(* Logix 5000 project; controller LeakTestAuto vendor 1 type 14 code 226 rev 37.11; software revision 37.01; part 6 of 13 *)
(* tags used below, declared in another part *)
   AOI_CTS1 : AOI_CTS_INSTRUMENT;
   AOI_OP220_HomingSeq : AOI_Sequencer_x64;
   AOI_OP220_Seq : AOI_Sequencer_x64;
   AOI_RobotPos : AOI_RobotPositions;
   AOI_SeqSteps : AOI_StandardSeqSteps;
   AOI_SRX100 : AOI_KeyenceBarcode;
   Barcode_ResultData : STR_Barcode;
   BarcodeBypass : BOOL;
   BarcodeInputs : udt_KeyenceScannerInputs;
   BarcodeScanner : udt_OutputStructure;
   Config_ConveyorHomeCounter : DINT;
   Config_ConveyorHomeCounterEnter : BOOL;
   Config_CylinderWaitTime : DINT;
   Config_CylinderWaitTimeEnter : BOOL;
   Config_MaxFailCount : DINT;
   Config_MaxFailCountEnter : BOOL;
   Conveyor : udt_OutputStructure;
   Conveyor_Seq : udt_SequenceStructure_X64;
   ConveyorHomeCounter : COUNTER;
   CTS1_BarcodeWrite : STRING80;
   CTS2_BarcodeWrite : STRING80;
   CurrentDUTData : udt_DUTHistory[2];
   DryCycle_N1Ready : BOOL;
   DryCycle_N2Ready : BOOL;
   FailCount : COUNTER;
   HomingClearNestsBypass : BOOL;
   InfeedCounter : COUNTER;
   LeakTester1 : udt_OutputStructure;
   LeakTester2 : udt_OutputStructure;
   Mode_CapCTS : BOOL;
   Nest1Bypass : BOOL;
   Nest1Cylinder : udt_OutputStructure;
   Nest1Empty : BOOL;
   Nest1Ready : BOOL;
   Nest2Bypass : BOOL;
   Nest2Cylinder : udt_OutputStructure;
   Nest2Empty : BOOL;
   Nest2Ready : BOOL;
   ONS_FailBinRemoved : BOOL;
   OP220 : udt_Mode;
   OP220_HomingSeq : udt_SequenceStructure_X64;
   OP220_Seq : udt_SequenceStructure_X64;
   OutfeedCounter : COUNTER;
   ResetFeedCounters : BOOL;
   RFID_CmdNest1 : BOOL;
   RFID_CmdNest2 : BOOL;
   RFID_Nest2Delay : TIMER;
   RFID_RWHAllPort : RWH_CMD;
   RFID_TagStatus : BOOL[32];
   RFIDBypass : BOOL;
   RFIDScanner : udt_OutputStructure;
   Robot : udt_OutputStructure;
   RobotGripper : udt_OutputStructure;
   RobotInputs : udt_EpsonInputs;
   RobotOutputs : udt_EpsonOutputs;
   TON_ConvUnloadDelay : TIMER;
   TON_FailChute : TIMER[10];
   TON_Nest1DryCycleDryTest : TIMER;
   TON_Nest2DryCycleDryTest : TIMER;
   I_OP220_N3_CONVEYOR_UNLOAD : ALIAS FOR Local:3:I.Pt14.Data;
   I_OP220_N3_DUT_PRE_NEST_0 : ALIAS FOR Local:3:I.Pt00.Data;
   I_OP220_N3_DUT_PRE_NEST_1 : ALIAS FOR Local:3:I.Pt01.Data;
   I_OP220_N3_DUT_PRE_NEST_2 : ALIAS FOR Local:3:I.Pt02.Data;
   I_OP220_N3_NEST1_EXTEND : ALIAS FOR Local:3:I.Pt04.Data;
   I_OP220_N3_NEST1_HOME : ALIAS FOR Local:3:I.Pt03.Data;
   I_OP220_N3_NEST2_EXTEND : ALIAS FOR Local:3:I.Pt06.Data;
   I_OP220_N3_NEST2_HOME : ALIAS FOR Local:3:I.Pt05.Data;
   I_OP220_N3_REJECT_BIN_OK : ALIAS FOR Local:3:I.Pt09.Data;
   I_OP220_N3_REJECT_CHUTE_PART : ALIAS FOR Local:3:I.Pt10.Data;
   James_Dint : DINT;   // James Test Word
   O_OP220_N5_CONV_REV : ALIAS FOR Local:5:O.Pt11.Data;
   O_OP220_N5_EN_MAIN_AIR : ALIAS FOR Local:5:O.Pt04.Data;
   O_OP220_N5_EN_ROBOT_LATCHOFF : ALIAS FOR Local:5:O.Pt09.Data;
   PLC : AOI_PLC;
   ST1_Ignition_SerialNum : STRING;
   ST2_Ignition_SerialNum : STRING;
(* MainProgram, continued *)

ROUTINE R06_IOControl   (* ladder *)
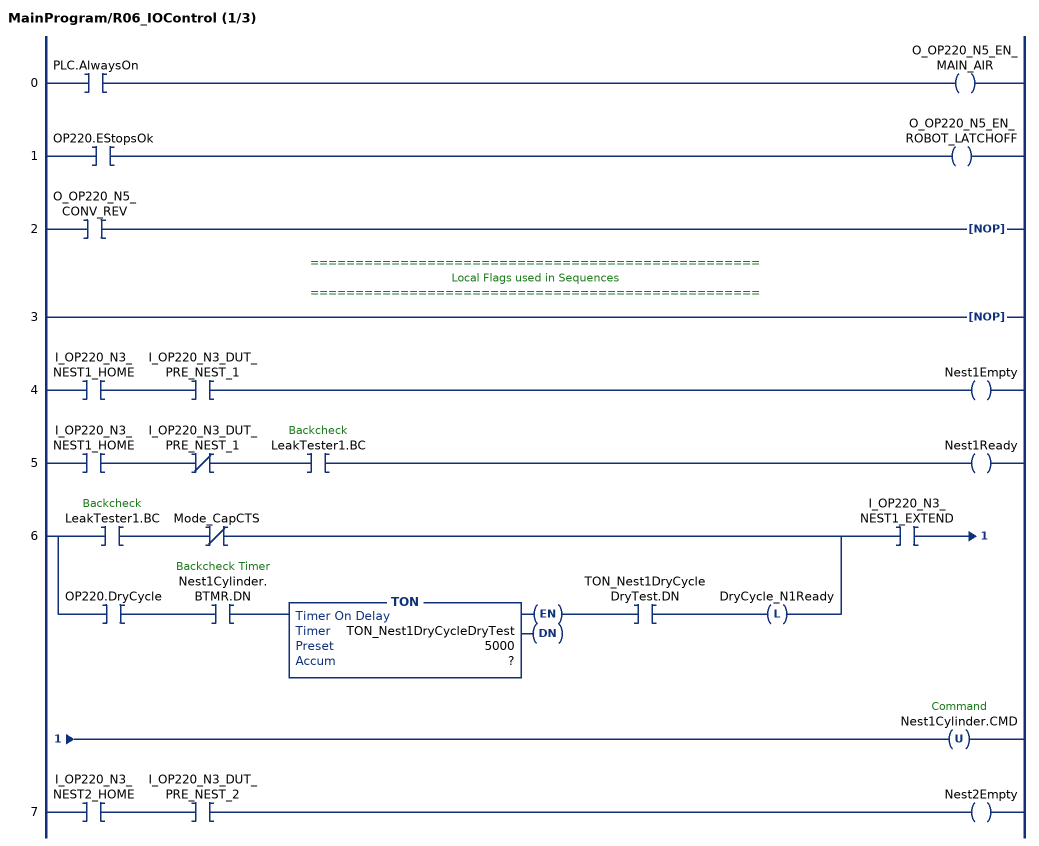
   0: XIC(PLC.AlwaysOn)OTE(O_OP220_N5_EN_MAIN_AIR);
   1: XIC(OP220.EStopsOk)OTE(O_OP220_N5_EN_ROBOT_LATCHOFF);
   2: XIC(O_OP220_N5_CONV_REV)NOP();
   // ==================================================
   // Local Flags used in Sequences
   // ==================================================
   3: NOP();
   4: XIC(I_OP220_N3_NEST1_HOME)XIC(I_OP220_N3_DUT_PRE_NEST_1)OTE(Nest1Empty);
   5: XIC(I_OP220_N3_NEST1_HOME)XIO(I_OP220_N3_DUT_PRE_NEST_1)XIC(LeakTester1.BC)OTE(Nest1Ready);
   6: [XIC(LeakTester1.BC) XIO(Mode_CapCTS) ,XIC(OP220.DryCycle) XIC(Nest1Cylinder.BTMR.DN) TON(TON_Nest1DryCycleDryTest,?,?) XIC(TON_Nest1DryCycleDryTest.DN) OTL(DryCycle_N1Ready) ]XIC(I_OP220_N3_NEST1_EXTEND)OTU(Nest1Cylinder.CMD);
   7: XIC(I_OP220_N3_NEST2_HOME)XIC(I_OP220_N3_DUT_PRE_NEST_2)OTE(Nest2Empty);
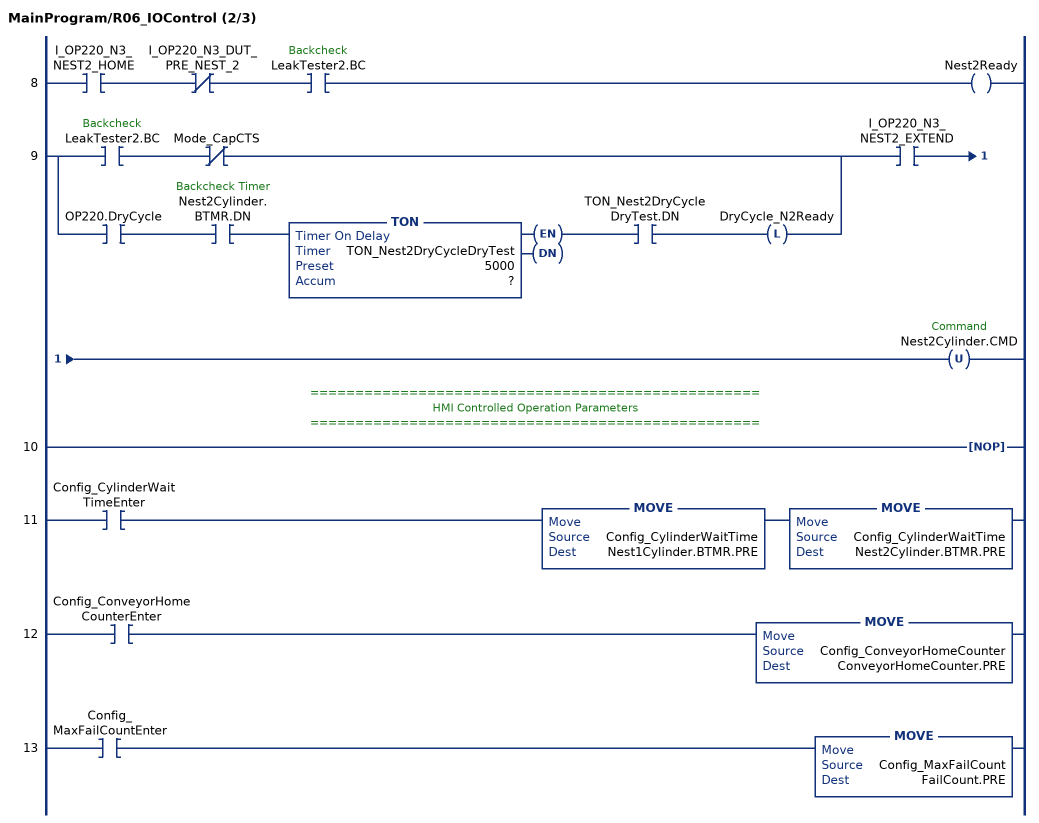
   8: XIC(I_OP220_N3_NEST2_HOME)XIO(I_OP220_N3_DUT_PRE_NEST_2)XIC(LeakTester2.BC)OTE(Nest2Ready);
   9: [XIC(LeakTester2.BC) XIO(Mode_CapCTS) ,XIC(OP220.DryCycle) XIC(Nest2Cylinder.BTMR.DN) TON(TON_Nest2DryCycleDryTest,?,?) XIC(TON_Nest2DryCycleDryTest.DN) OTL(DryCycle_N2Ready) ]XIC(I_OP220_N3_NEST2_EXTEND)OTU(Nest2Cylinder.CMD);
   // ==================================================
   // HMI Controlled Operation Parameters
   // ==================================================
   10: NOP();
   11: XIC(Config_CylinderWaitTimeEnter)MOVE(Config_CylinderWaitTime,Nest1Cylinder.BTMR.PRE)MOVE(Config_CylinderWaitTime,Nest2Cylinder.BTMR.PRE);
   12: XIC(Config_ConveyorHomeCounterEnter)MOVE(Config_ConveyorHomeCounter,ConveyorHomeCounter.PRE);
   13: XIC(Config_MaxFailCountEnter)MOVE(Config_MaxFailCount,FailCount.PRE);
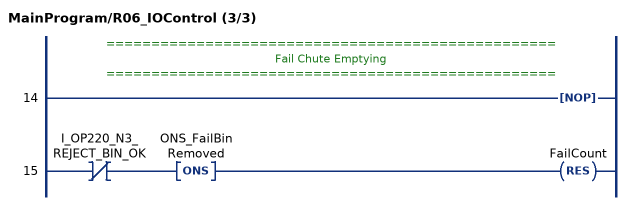
   // ==================================================
   // Fail Chute Emptying
   // ==================================================
   14: NOP();
   15: XIO(I_OP220_N3_REJECT_BIN_OK)ONS(ONS_FailBinRemoved)RES(FailCount);
END_ROUTINE

ROUTINE R09_Homing   (* ladder *)
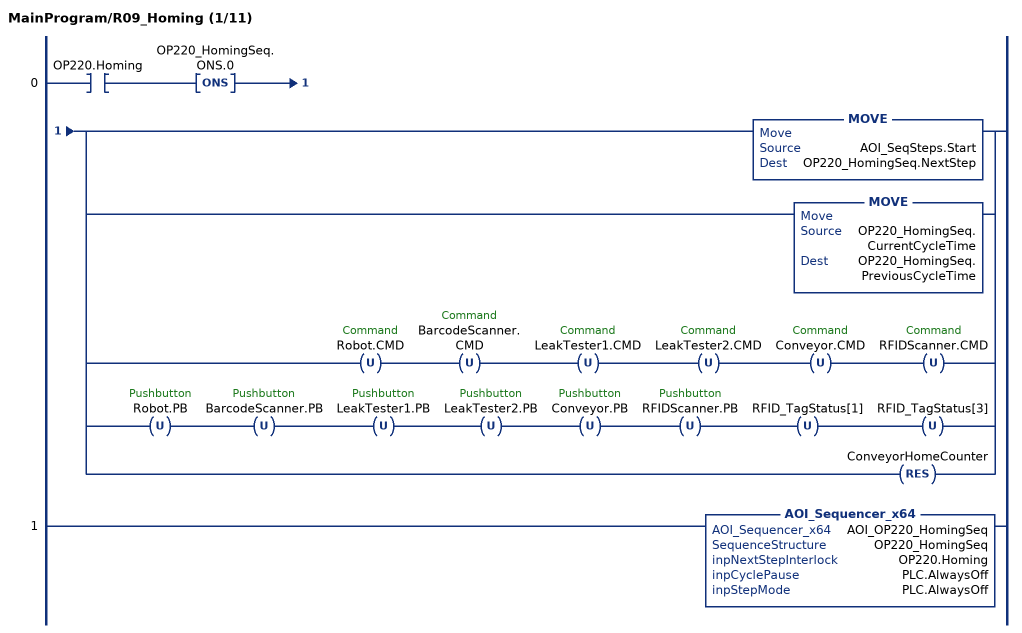
   0: XIC(OP220.Homing)ONS(OP220_HomingSeq.ONS.0)[MOVE(AOI_SeqSteps.Start,OP220_HomingSeq.NextStep) ,MOVE(OP220_HomingSeq.CurrentCycleTime,OP220_HomingSeq.PreviousCycleTime) ,OTU(Robot.CMD) OTU(BarcodeScanner.CMD) OTU(LeakTester1.CMD) OTU(LeakTester2.CMD) OTU(Conveyor.CMD) OTU(RFIDScanner.CMD) ,OTU(Robot.PB) OTU(BarcodeScanner.PB) OTU(LeakTester1.PB) OTU(LeakTester2.PB) OTU(Conveyor.PB) OTU(RFIDScanner.PB) OTU(RFID_TagStatus[1]) OTU(RFID_TagStatus[3]) ,RES(ConveyorHomeCounter) ];
   1: AOI_Sequencer_x64(AOI_OP220_HomingSeq,OP220_HomingSeq,OP220.Homing,PLC.AlwaysOff,PLC.AlwaysOff);
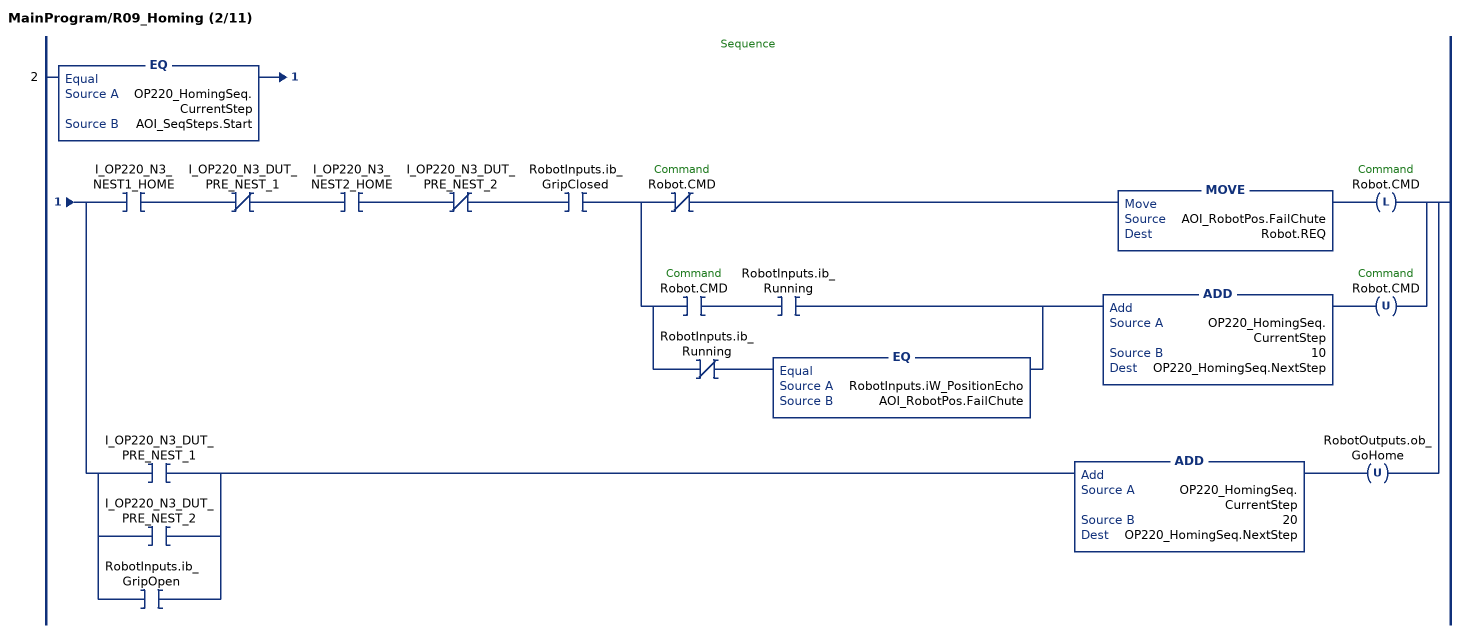
   // Sequence
   2: EQ(OP220_HomingSeq.CurrentStep,AOI_SeqSteps.Start)[XIC(I_OP220_N3_NEST1_HOME) XIO(I_OP220_N3_DUT_PRE_NEST_1) XIC(I_OP220_N3_NEST2_HOME) XIO(I_OP220_N3_DUT_PRE_NEST_2) XIC(RobotInputs.ib_GripClosed) [XIO(Robot.CMD) MOVE(AOI_RobotPos.FailChute,Robot.REQ) OTL(Robot.CMD) ,[XIC(Robot.CMD) XIC(RobotInputs.ib_Running) ,XIO(RobotInputs.ib_Running) EQ(RobotInputs.iW_PositionEcho,AOI_RobotPos.FailChute) ] ADD(OP220_HomingSeq.CurrentStep,10,OP220_HomingSeq.NextStep) OTU(Robot.CMD) ] ,[XIC(I_OP220_N3_DUT_PRE_NEST_1) ,XIC(I_OP220_N3_DUT_PRE_NEST_2) ,XIC(RobotInputs.ib_GripOpen) ] ADD(OP220_HomingSeq.CurrentStep,20,OP220_HomingSeq.NextStep) OTU(RobotOutputs.ob_GoHome) ];
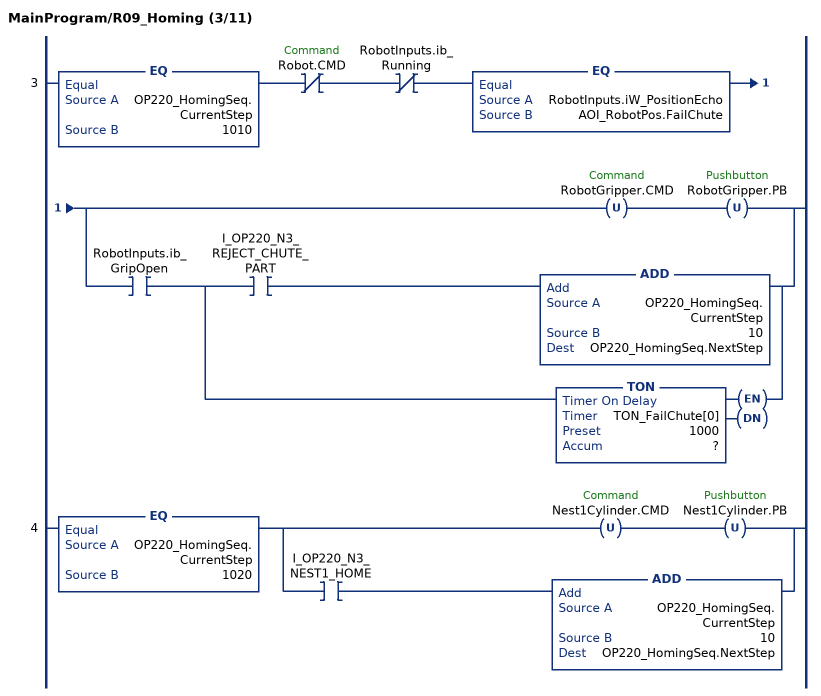
   3: EQ(OP220_HomingSeq.CurrentStep,1010)XIO(Robot.CMD)XIO(RobotInputs.ib_Running)EQ(RobotInputs.iW_PositionEcho,AOI_RobotPos.FailChute)[OTU(RobotGripper.CMD) OTU(RobotGripper.PB) ,XIC(RobotInputs.ib_GripOpen) [XIC(I_OP220_N3_REJECT_CHUTE_PART) ADD(OP220_HomingSeq.CurrentStep,10,OP220_HomingSeq.NextStep) ,TON(TON_FailChute[0],?,?) ] ];
   4: EQ(OP220_HomingSeq.CurrentStep,1020)[OTU(Nest1Cylinder.CMD) OTU(Nest1Cylinder.PB) ,XIC(I_OP220_N3_NEST1_HOME) ADD(OP220_HomingSeq.CurrentStep,10,OP220_HomingSeq.NextStep) ];
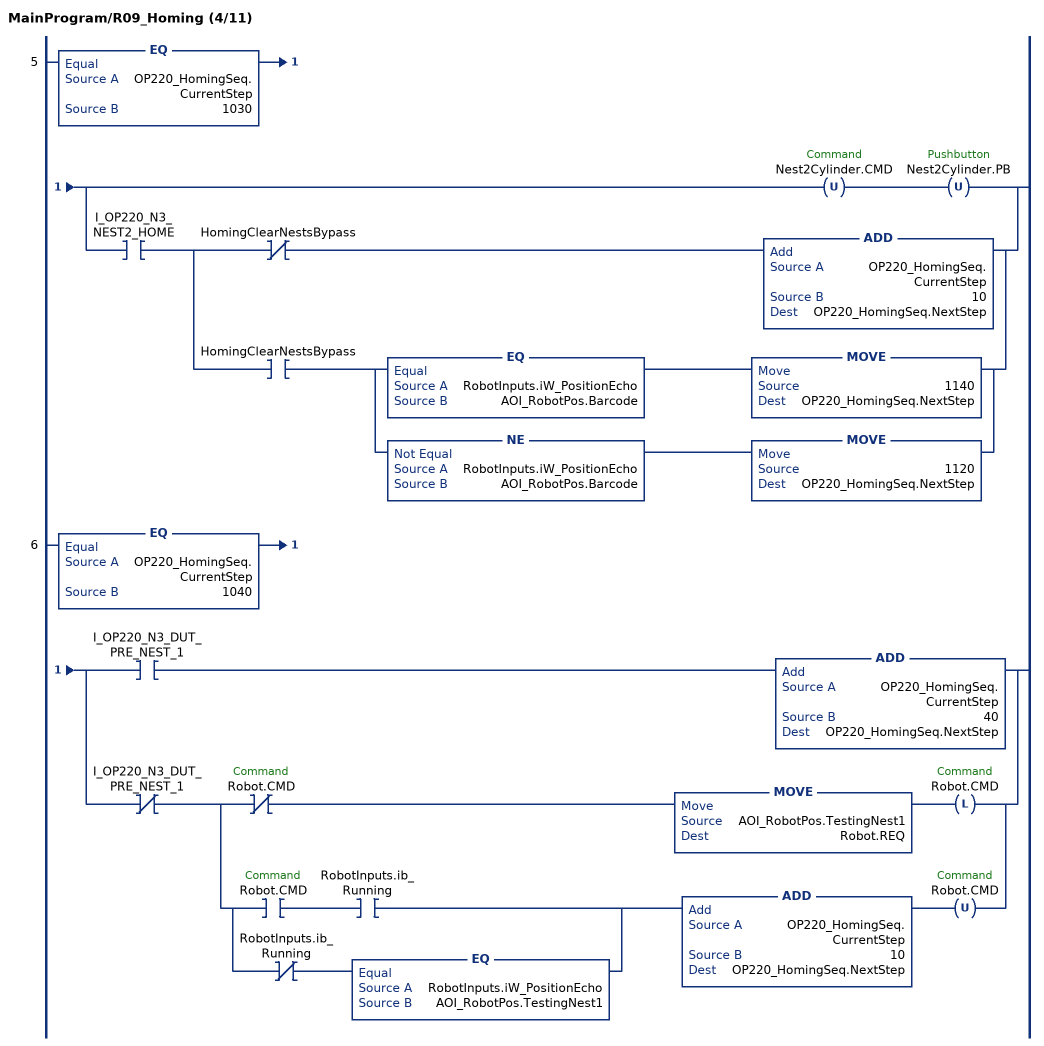
   5: EQ(OP220_HomingSeq.CurrentStep,1030)[OTU(Nest2Cylinder.CMD) OTU(Nest2Cylinder.PB) ,XIC(I_OP220_N3_NEST2_HOME) [XIO(HomingClearNestsBypass) ADD(OP220_HomingSeq.CurrentStep,10,OP220_HomingSeq.NextStep) ,XIC(HomingClearNestsBypass) [EQ(RobotInputs.iW_PositionEcho,AOI_RobotPos.Barcode) MOVE(1140,OP220_HomingSeq.NextStep) ,NE(RobotInputs.iW_PositionEcho,AOI_RobotPos.Barcode) MOVE(1120,OP220_HomingSeq.NextStep) ] ] ];
   6: EQ(OP220_HomingSeq.CurrentStep,1040)[XIC(I_OP220_N3_DUT_PRE_NEST_1) ADD(OP220_HomingSeq.CurrentStep,40,OP220_HomingSeq.NextStep) ,XIO(I_OP220_N3_DUT_PRE_NEST_1) [XIO(Robot.CMD) MOVE(AOI_RobotPos.TestingNest1,Robot.REQ) OTL(Robot.CMD) ,[XIC(Robot.CMD) XIC(RobotInputs.ib_Running) ,XIO(RobotInputs.ib_Running) EQ(RobotInputs.iW_PositionEcho,AOI_RobotPos.TestingNest1) ] ADD(OP220_HomingSeq.CurrentStep,10,OP220_HomingSeq.NextStep) OTU(Robot.CMD) ] ];
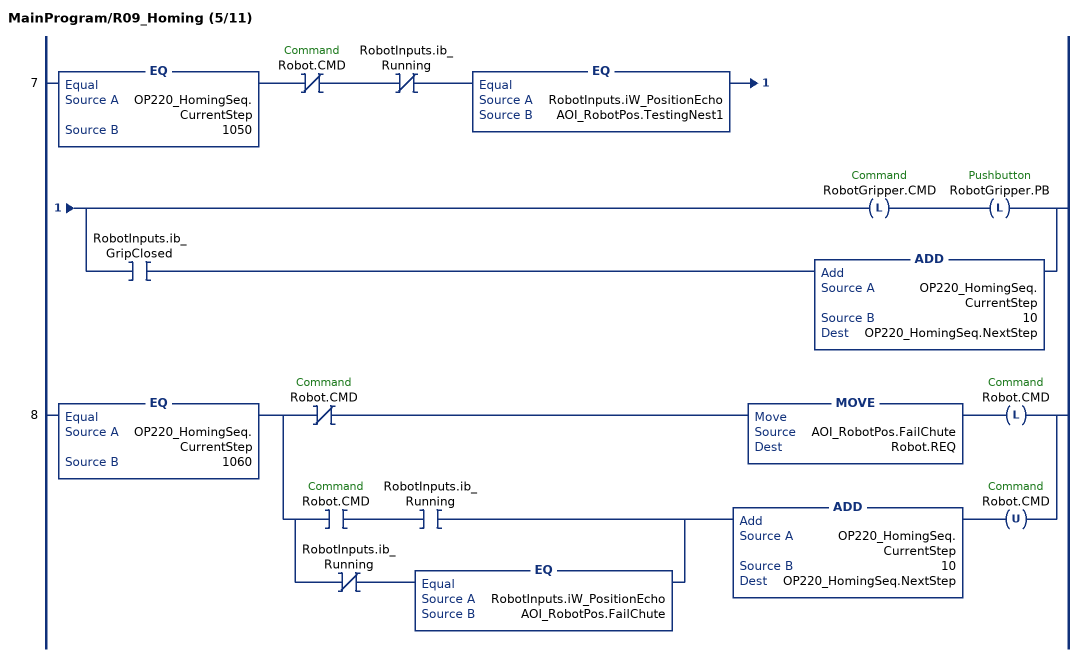
   7: EQ(OP220_HomingSeq.CurrentStep,1050)XIO(Robot.CMD)XIO(RobotInputs.ib_Running)EQ(RobotInputs.iW_PositionEcho,AOI_RobotPos.TestingNest1)[OTL(RobotGripper.CMD) OTL(RobotGripper.PB) ,XIC(RobotInputs.ib_GripClosed) ADD(OP220_HomingSeq.CurrentStep,10,OP220_HomingSeq.NextStep) ];
   8: EQ(OP220_HomingSeq.CurrentStep,1060)[XIO(Robot.CMD) MOVE(AOI_RobotPos.FailChute,Robot.REQ) OTL(Robot.CMD) ,[XIC(Robot.CMD) XIC(RobotInputs.ib_Running) ,XIO(RobotInputs.ib_Running) EQ(RobotInputs.iW_PositionEcho,AOI_RobotPos.FailChute) ] ADD(OP220_HomingSeq.CurrentStep,10,OP220_HomingSeq.NextStep) OTU(Robot.CMD) ];
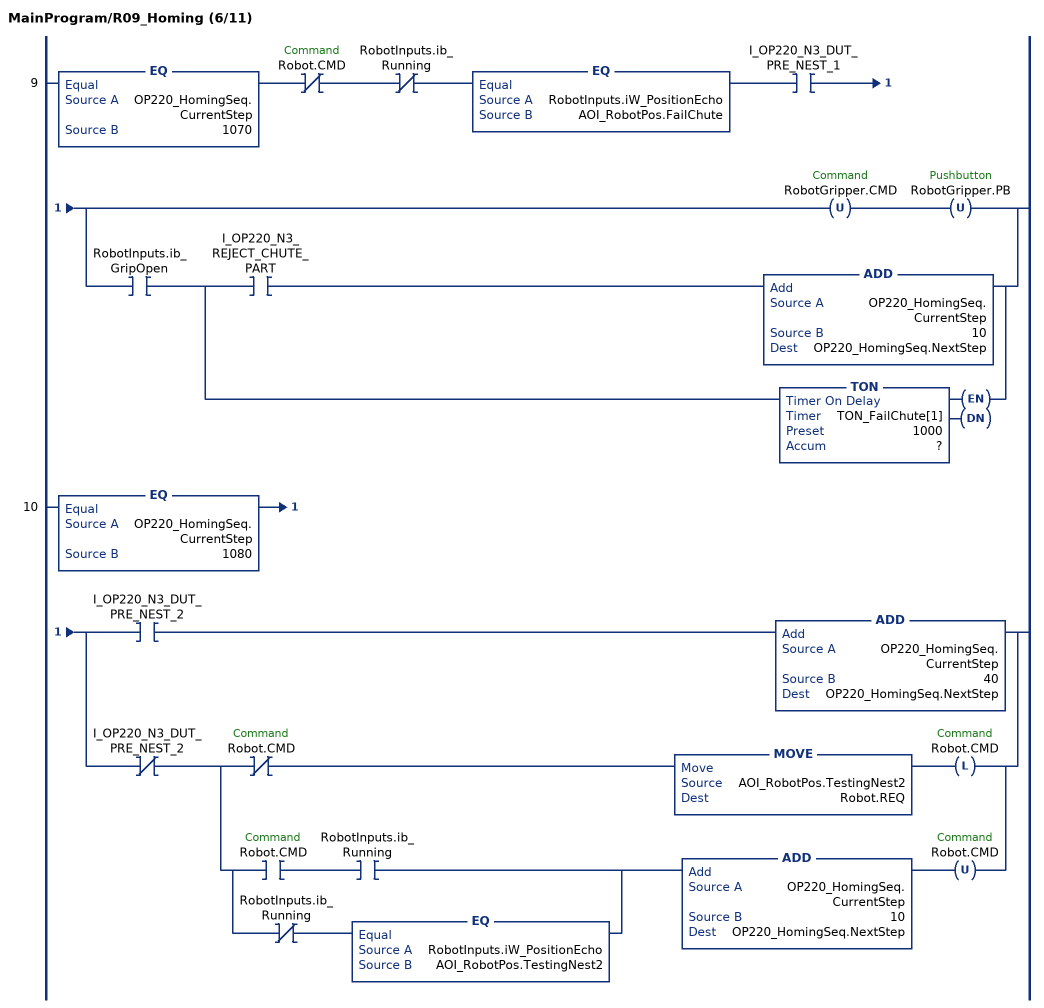
   9: EQ(OP220_HomingSeq.CurrentStep,1070)XIO(Robot.CMD)XIO(RobotInputs.ib_Running)EQ(RobotInputs.iW_PositionEcho,AOI_RobotPos.FailChute)XIC(I_OP220_N3_DUT_PRE_NEST_1)[OTU(RobotGripper.CMD) OTU(RobotGripper.PB) ,XIC(RobotInputs.ib_GripOpen) [XIC(I_OP220_N3_REJECT_CHUTE_PART) ADD(OP220_HomingSeq.CurrentStep,10,OP220_HomingSeq.NextStep) ,TON(TON_FailChute[1],?,?) ] ];
   10: EQ(OP220_HomingSeq.CurrentStep,1080)[XIC(I_OP220_N3_DUT_PRE_NEST_2) ADD(OP220_HomingSeq.CurrentStep,40,OP220_HomingSeq.NextStep) ,XIO(I_OP220_N3_DUT_PRE_NEST_2) [XIO(Robot.CMD) MOVE(AOI_RobotPos.TestingNest2,Robot.REQ) OTL(Robot.CMD) ,[XIC(Robot.CMD) XIC(RobotInputs.ib_Running) ,XIO(RobotInputs.ib_Running) EQ(RobotInputs.iW_PositionEcho,AOI_RobotPos.TestingNest2) ] ADD(OP220_HomingSeq.CurrentStep,10,OP220_HomingSeq.NextStep) OTU(Robot.CMD) ] ];
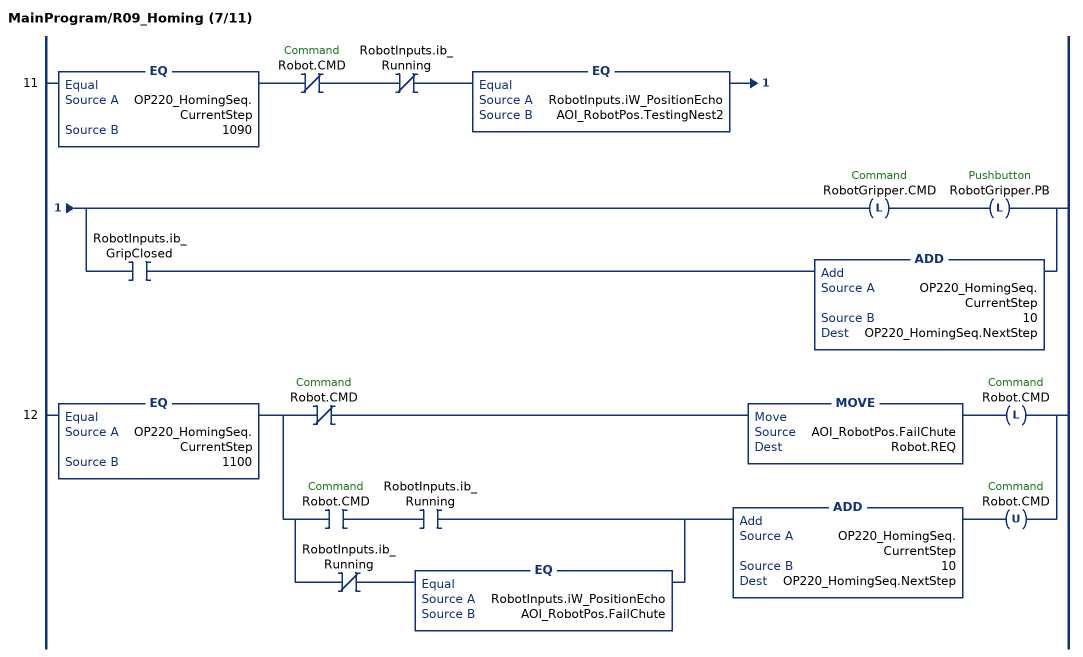
   11: EQ(OP220_HomingSeq.CurrentStep,1090)XIO(Robot.CMD)XIO(RobotInputs.ib_Running)EQ(RobotInputs.iW_PositionEcho,AOI_RobotPos.TestingNest2)[OTL(RobotGripper.CMD) OTL(RobotGripper.PB) ,XIC(RobotInputs.ib_GripClosed) ADD(OP220_HomingSeq.CurrentStep,10,OP220_HomingSeq.NextStep) ];
   12: EQ(OP220_HomingSeq.CurrentStep,1100)[XIO(Robot.CMD) MOVE(AOI_RobotPos.FailChute,Robot.REQ) OTL(Robot.CMD) ,[XIC(Robot.CMD) XIC(RobotInputs.ib_Running) ,XIO(RobotInputs.ib_Running) EQ(RobotInputs.iW_PositionEcho,AOI_RobotPos.FailChute) ] ADD(OP220_HomingSeq.CurrentStep,10,OP220_HomingSeq.NextStep) OTU(Robot.CMD) ];
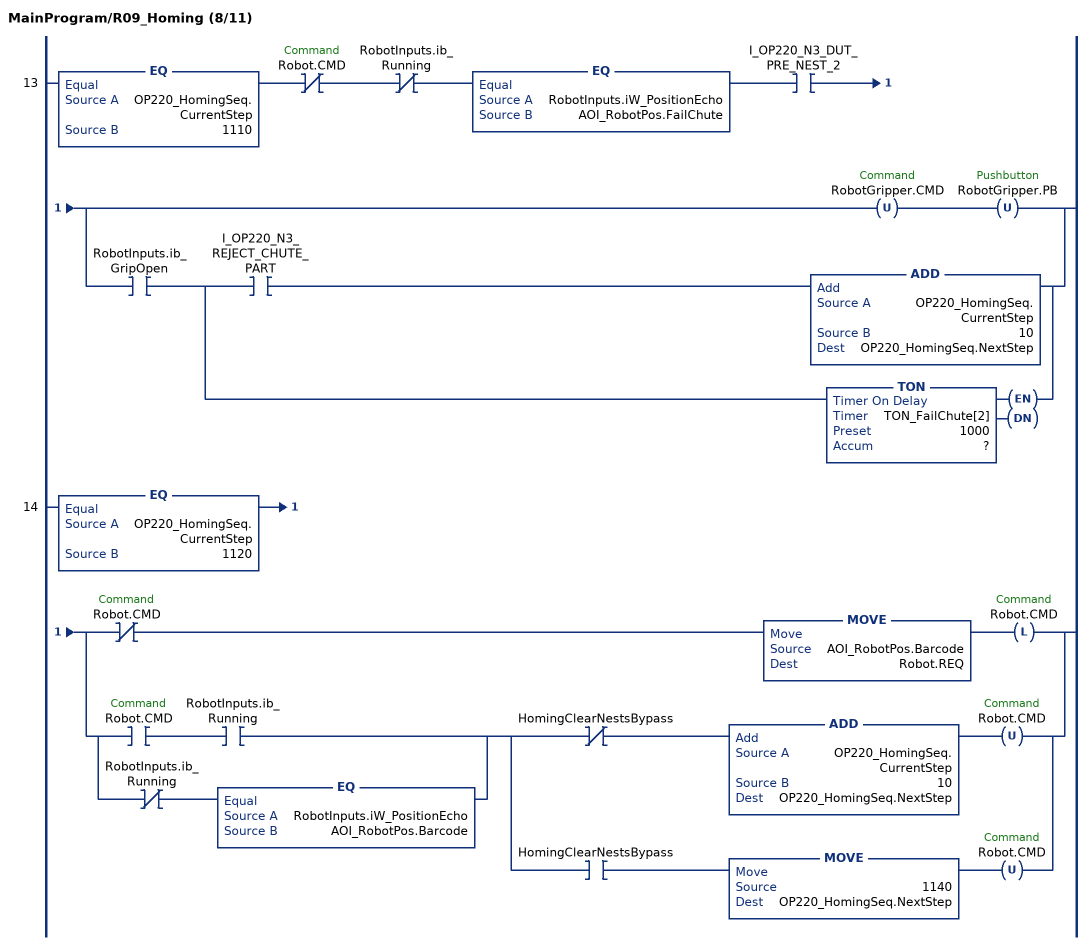
   13: EQ(OP220_HomingSeq.CurrentStep,1110)XIO(Robot.CMD)XIO(RobotInputs.ib_Running)EQ(RobotInputs.iW_PositionEcho,AOI_RobotPos.FailChute)XIC(I_OP220_N3_DUT_PRE_NEST_2)[OTU(RobotGripper.CMD) OTU(RobotGripper.PB) ,XIC(RobotInputs.ib_GripOpen) [XIC(I_OP220_N3_REJECT_CHUTE_PART) ADD(OP220_HomingSeq.CurrentStep,10,OP220_HomingSeq.NextStep) ,TON(TON_FailChute[2],?,?) ] ];
   14: EQ(OP220_HomingSeq.CurrentStep,1120)[XIO(Robot.CMD) MOVE(AOI_RobotPos.Barcode,Robot.REQ) OTL(Robot.CMD) ,[XIC(Robot.CMD) XIC(RobotInputs.ib_Running) ,XIO(RobotInputs.ib_Running) EQ(RobotInputs.iW_PositionEcho,AOI_RobotPos.Barcode) ] [XIO(HomingClearNestsBypass) ADD(OP220_HomingSeq.CurrentStep,10,OP220_HomingSeq.NextStep) OTU(Robot.CMD) ,XIC(HomingClearNestsBypass) MOVE(1140,OP220_HomingSeq.NextStep) OTU(Robot.CMD) ] ];
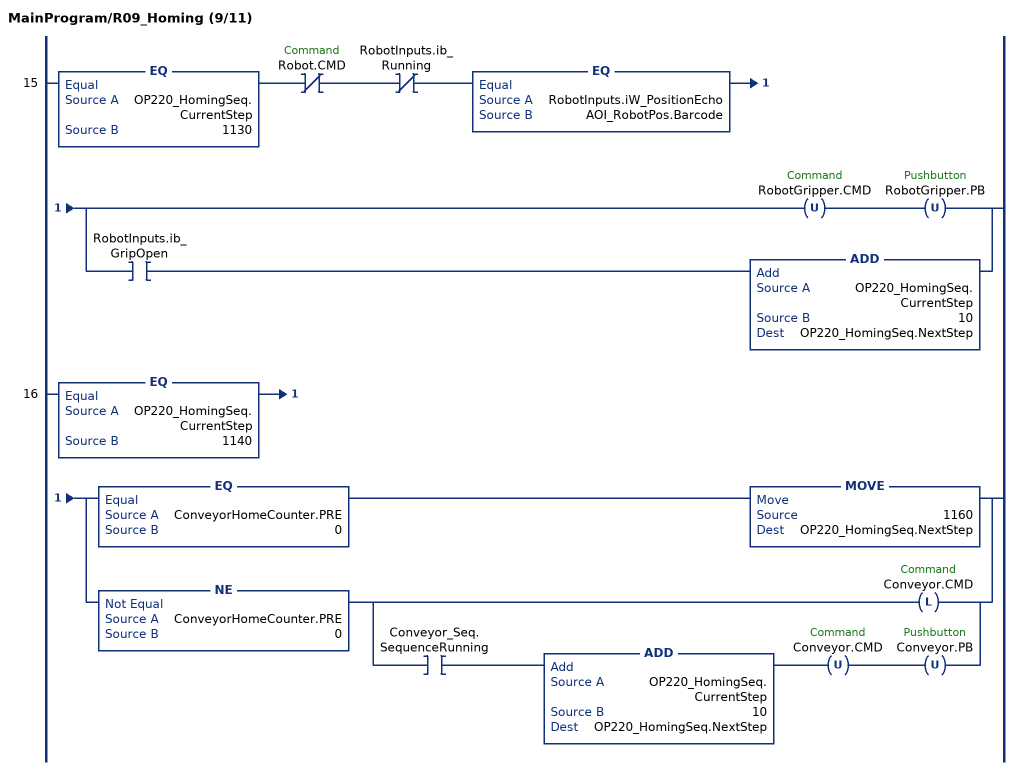
   15: EQ(OP220_HomingSeq.CurrentStep,1130)XIO(Robot.CMD)XIO(RobotInputs.ib_Running)EQ(RobotInputs.iW_PositionEcho,AOI_RobotPos.Barcode)[OTU(RobotGripper.CMD) OTU(RobotGripper.PB) ,XIC(RobotInputs.ib_GripOpen) ADD(OP220_HomingSeq.CurrentStep,10,OP220_HomingSeq.NextStep) ];
   16: EQ(OP220_HomingSeq.CurrentStep,1140)[EQ(ConveyorHomeCounter.PRE,0) MOVE(1160,OP220_HomingSeq.NextStep) ,NE(ConveyorHomeCounter.PRE,0) [OTL(Conveyor.CMD) ,XIC(Conveyor_Seq.SequenceRunning) ADD(OP220_HomingSeq.CurrentStep,10,OP220_HomingSeq.NextStep) OTU(Conveyor.CMD) OTU(Conveyor.PB) ] ];
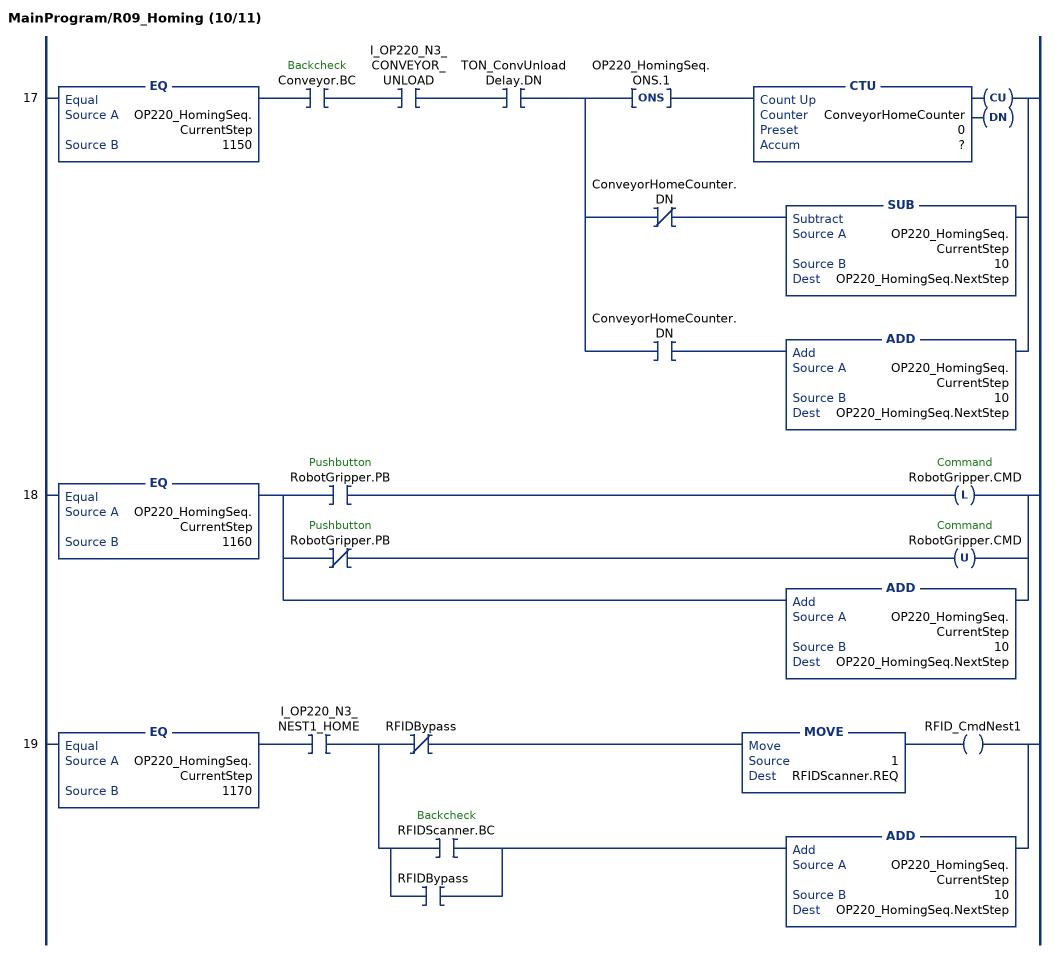
   17: EQ(OP220_HomingSeq.CurrentStep,1150)XIC(Conveyor.BC)XIC(I_OP220_N3_CONVEYOR_UNLOAD)XIC(TON_ConvUnloadDelay.DN)[ONS(OP220_HomingSeq.ONS.1) CTU(ConveyorHomeCounter,?,?) ,[XIO(ConveyorHomeCounter.DN) SUB(OP220_HomingSeq.CurrentStep,10,OP220_HomingSeq.NextStep) ,XIC(ConveyorHomeCounter.DN) ADD(OP220_HomingSeq.CurrentStep,10,OP220_HomingSeq.NextStep) ] ];
   18: EQ(OP220_HomingSeq.CurrentStep,1160)[XIC(RobotGripper.PB) OTL(RobotGripper.CMD) ,XIO(RobotGripper.PB) OTU(RobotGripper.CMD) ,ADD(OP220_HomingSeq.CurrentStep,10,OP220_HomingSeq.NextStep) ];
   19: EQ(OP220_HomingSeq.CurrentStep,1170)XIC(I_OP220_N3_NEST1_HOME)[XIO(RFIDBypass) MOVE(1,RFIDScanner.REQ) OTE(RFID_CmdNest1) ,[XIC(RFIDScanner.BC) ,XIC(RFIDBypass) ] ADD(OP220_HomingSeq.CurrentStep,10,OP220_HomingSeq.NextStep) ];
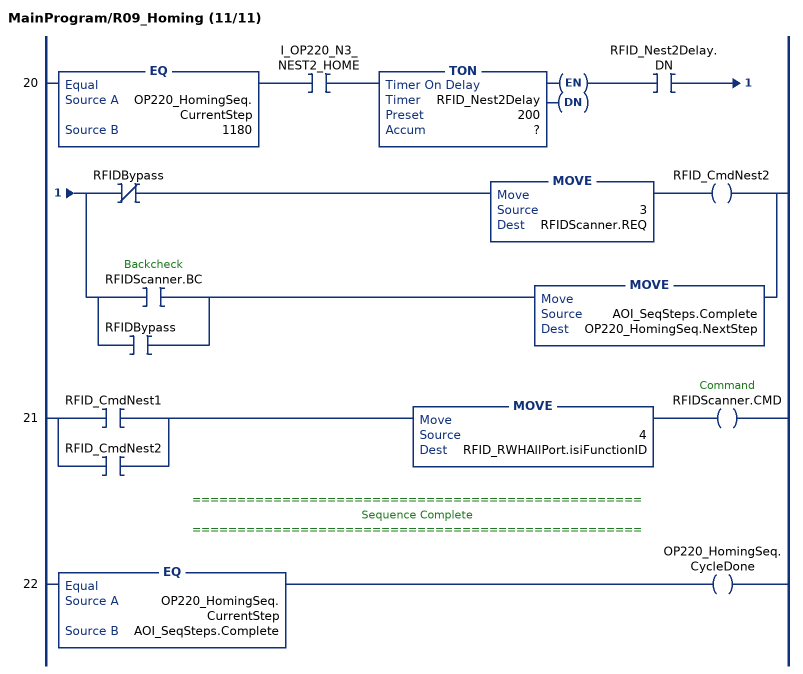
   20: EQ(OP220_HomingSeq.CurrentStep,1180)XIC(I_OP220_N3_NEST2_HOME)TON(RFID_Nest2Delay,?,?)XIC(RFID_Nest2Delay.DN)[XIO(RFIDBypass) MOVE(3,RFIDScanner.REQ) OTE(RFID_CmdNest2) ,[XIC(RFIDScanner.BC) ,XIC(RFIDBypass) ] MOVE(AOI_SeqSteps.Complete,OP220_HomingSeq.NextStep) ];
   21: [XIC(RFID_CmdNest1) ,XIC(RFID_CmdNest2) ]MOVE(4,RFID_RWHAllPort.isiFunctionID)OTE(RFIDScanner.CMD);
   // ==================================================
   // Sequence Complete
   // ==================================================
   22: EQ(OP220_HomingSeq.CurrentStep,AOI_SeqSteps.Complete)OTE(OP220_HomingSeq.CycleDone);
END_ROUTINE

ROUTINE R10_Sequence   (* ladder *)
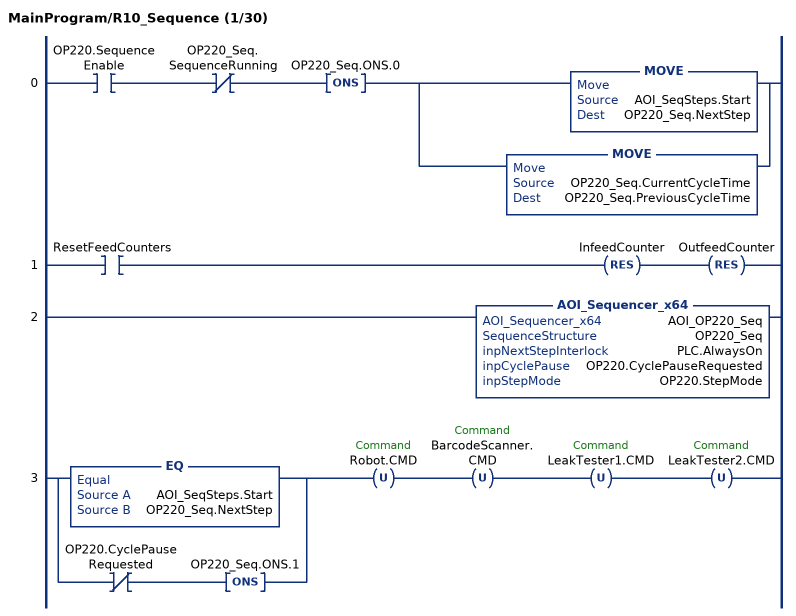
   0: XIC(OP220.SequenceEnable)XIO(OP220_Seq.SequenceRunning)ONS(OP220_Seq.ONS.0)[MOVE(AOI_SeqSteps.Start,OP220_Seq.NextStep) ,MOVE(OP220_Seq.CurrentCycleTime,OP220_Seq.PreviousCycleTime) ];
   1: XIC(ResetFeedCounters)RES(InfeedCounter)RES(OutfeedCounter);
   2: AOI_Sequencer_x64(AOI_OP220_Seq,OP220_Seq,PLC.AlwaysOn,OP220.CyclePauseRequested,OP220.StepMode);
   3: [EQ(AOI_SeqSteps.Start,OP220_Seq.NextStep) ,XIO(OP220.CyclePauseRequested) ONS(OP220_Seq.ONS.1) ]OTU(Robot.CMD)OTU(BarcodeScanner.CMD)OTU(LeakTester1.CMD)OTU(LeakTester2.CMD);
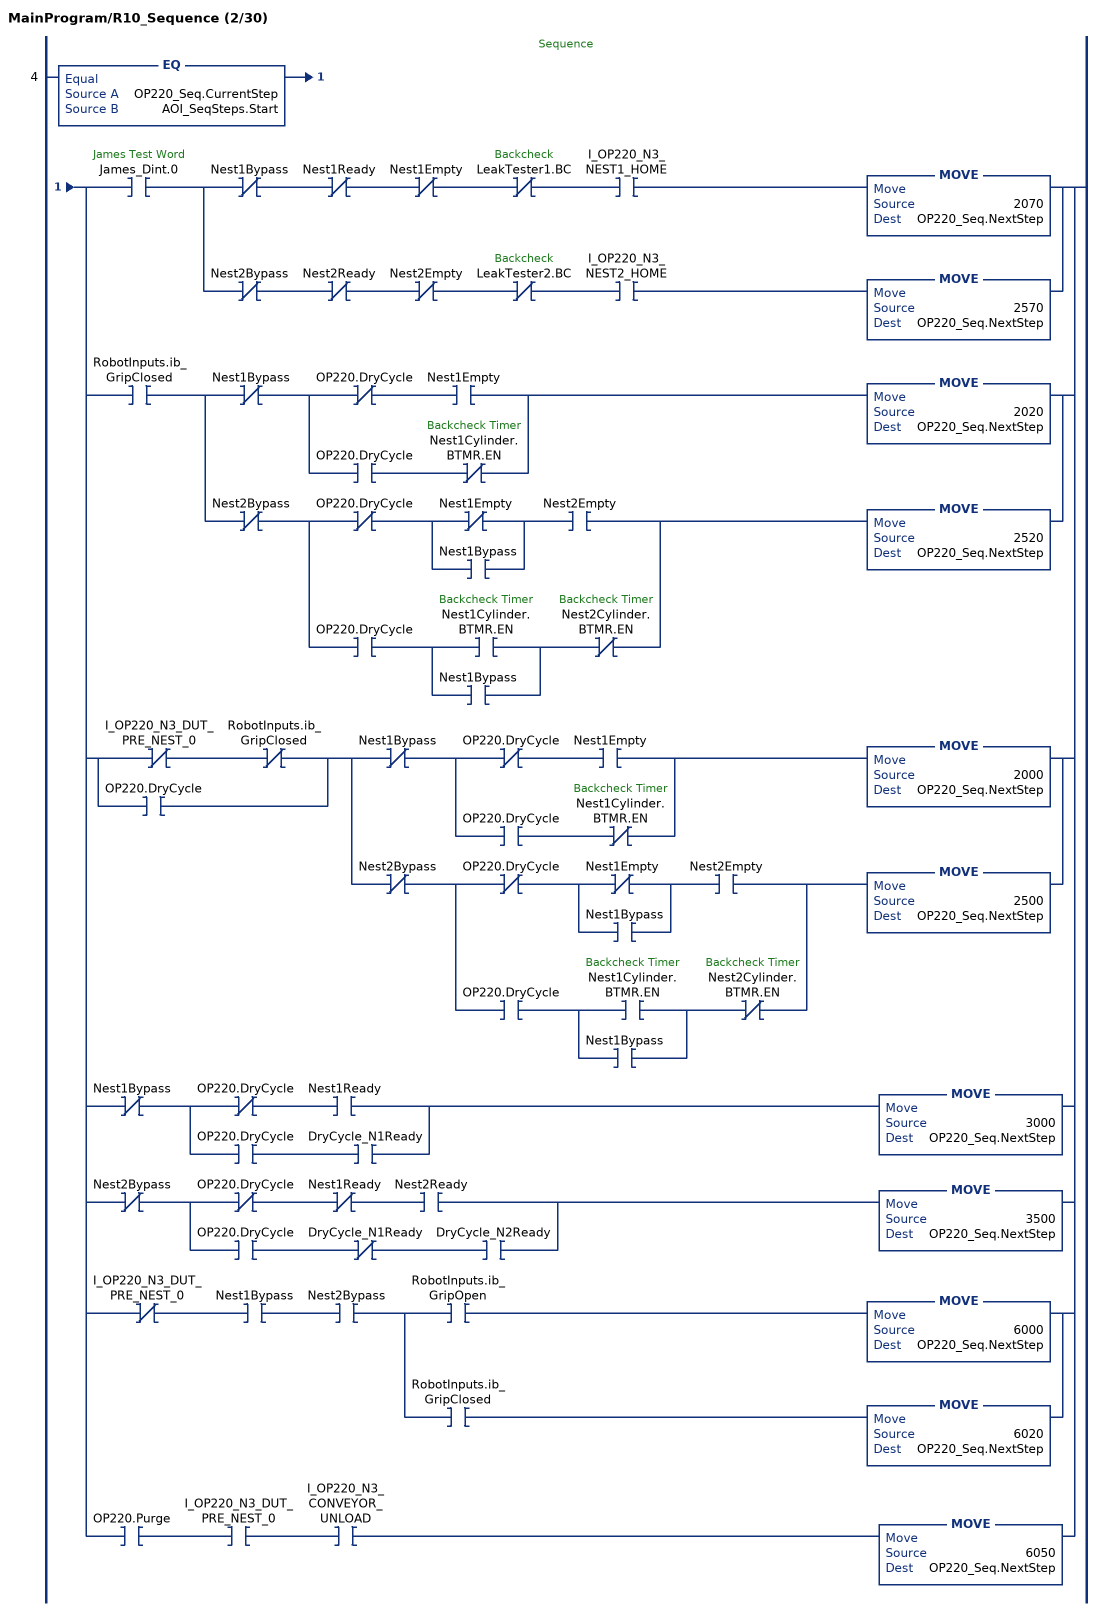
   // Sequence
   4: EQ(OP220_Seq.CurrentStep,AOI_SeqSteps.Start)[XIC(James_Dint.0) [XIO(Nest1Bypass) XIO(Nest1Ready) XIO(Nest1Empty) XIO(LeakTester1.BC) XIC(I_OP220_N3_NEST1_HOME) MOVE(2070,OP220_Seq.NextStep) ,XIO(Nest2Bypass) XIO(Nest2Ready) XIO(Nest2Empty) XIO(LeakTester2.BC) XIC(I_OP220_N3_NEST2_HOME) MOVE(2570,OP220_Seq.NextStep) ] ,XIC(RobotInputs.ib_GripClosed) [XIO(Nest1Bypass) [XIO(OP220.DryCycle) XIC(Nest1Empty) ,XIC(OP220.DryCycle) XIO(Nest1Cylinder.BTMR.EN) ] MOVE(2020,OP220_Seq.NextStep) ,XIO(Nest2Bypass) [XIO(OP220.DryCycle) [XIO(Nest1Empty) ,XIC(Nest1Bypass) ] XIC(Nest2Empty) ,XIC(OP220.DryCycle) [XIC(Nest1Cylinder.BTMR.EN) ,XIC(Nest1Bypass) ] XIO(Nest2Cylinder.BTMR.EN) ] MOVE(2520,OP220_Seq.NextStep) ] ,[XIO(I_OP220_N3_DUT_PRE_NEST_0) XIO(RobotInputs.ib_GripClosed) ,XIC(OP220.DryCycle) ] [XIO(Nest1Bypass) [XIO(OP220.DryCycle) XIC(Nest1Empty) ,XIC(OP220.DryCycle) XIO(Nest1Cylinder.BTMR.EN) ] MOVE(2000,OP220_Seq.NextStep) ,XIO(Nest2Bypass) [XIO(OP220.DryCycle) [XIO(Nest1Empty) ,XIC(Nest1Bypass) ] XIC(Nest2Empty) ,XIC(OP220.DryCycle) [XIC(Nest1Cylinder.BTMR.EN) ,XIC(Nest1Bypass) ] XIO(Nest2Cylinder.BTMR.EN) ] MOVE(2500,OP220_Seq.NextStep) ] ,[XIO(Nest1Bypass) [XIO(OP220.DryCycle) XIC(Nest1Ready) ,XIC(OP220.DryCycle) XIC(DryCycle_N1Ready) ] MOVE(3000,OP220_Seq.NextStep) ,XIO(Nest2Bypass) [XIO(OP220.DryCycle) XIO(Nest1Ready) XIC(Nest2Ready) ,XIC(OP220.DryCycle) XIO(DryCycle_N1Ready) XIC(DryCycle_N2Ready) ] MOVE(3500,OP220_Seq.NextStep) ] ,XIO(I_OP220_N3_DUT_PRE_NEST_0) XIC(Nest1Bypass) XIC(Nest2Bypass) [XIC(RobotInputs.ib_GripOpen) MOVE(6000,OP220_Seq.NextStep) ,XIC(RobotInputs.ib_GripClosed) MOVE(6020,OP220_Seq.NextStep) ] ,XIC(OP220.Purge) XIC(I_OP220_N3_DUT_PRE_NEST_0) XIC(I_OP220_N3_CONVEYOR_UNLOAD) MOVE(6050,OP220_Seq.NextStep) ];
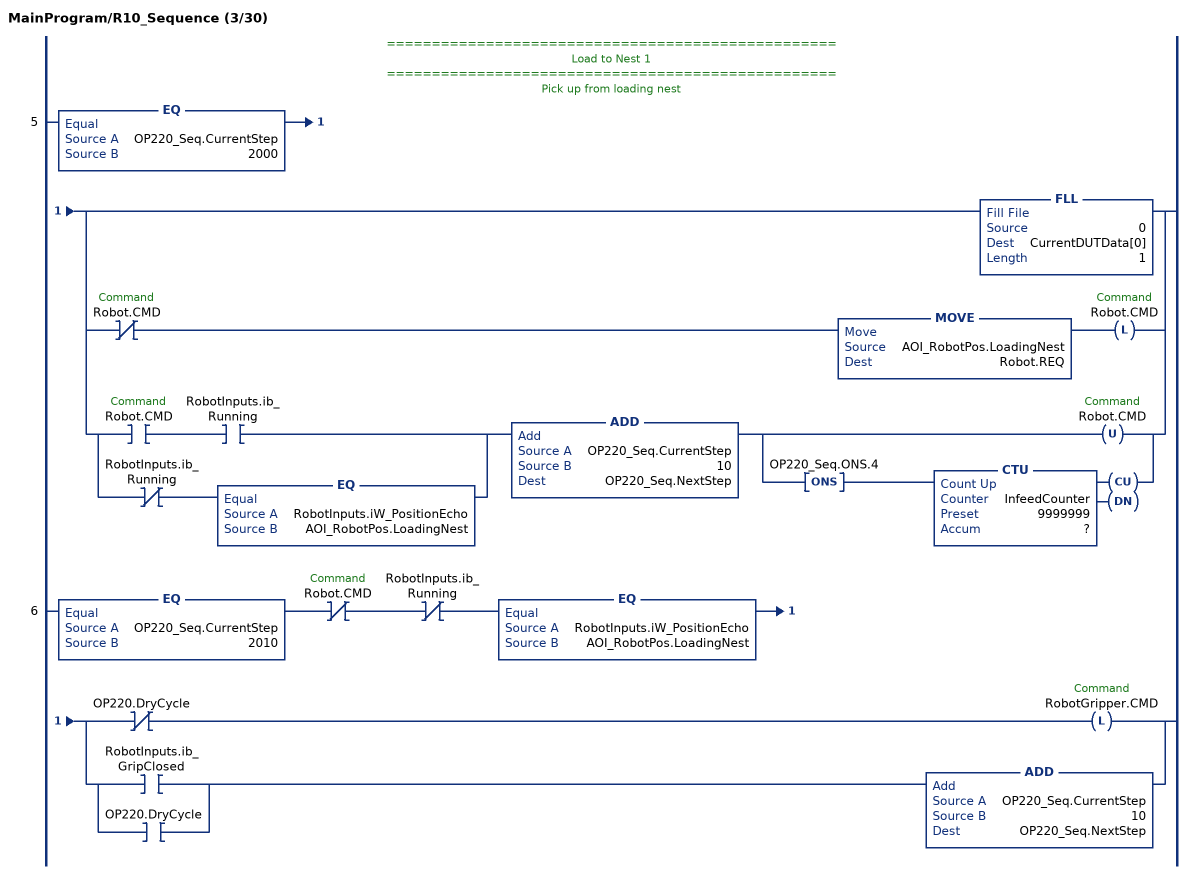
   // ==================================================
   // Load to Nest 1
   // ==================================================
   // Pick up from loading nest
   5: EQ(OP220_Seq.CurrentStep,2000)[FLL(0,CurrentDUTData[0],1) ,XIO(Robot.CMD) MOVE(AOI_RobotPos.LoadingNest,Robot.REQ) OTL(Robot.CMD) ,[XIC(Robot.CMD) XIC(RobotInputs.ib_Running) ,XIO(RobotInputs.ib_Running) EQ(RobotInputs.iW_PositionEcho,AOI_RobotPos.LoadingNest) ] ADD(OP220_Seq.CurrentStep,10,OP220_Seq.NextStep) [OTU(Robot.CMD) ,ONS(OP220_Seq.ONS.4) CTU(InfeedCounter,?,?) ] ];
   6: EQ(OP220_Seq.CurrentStep,2010)XIO(Robot.CMD)XIO(RobotInputs.ib_Running)EQ(RobotInputs.iW_PositionEcho,AOI_RobotPos.LoadingNest)[XIO(OP220.DryCycle) OTL(RobotGripper.CMD) ,[XIC(RobotInputs.ib_GripClosed) ,XIC(OP220.DryCycle) ] ADD(OP220_Seq.CurrentStep,10,OP220_Seq.NextStep) ];
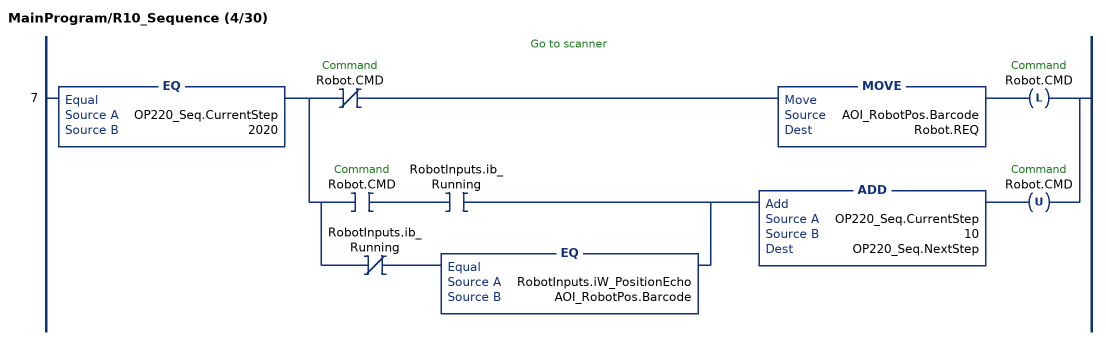
   // Go to scanner
   7: EQ(OP220_Seq.CurrentStep,2020)[XIO(Robot.CMD) MOVE(AOI_RobotPos.Barcode,Robot.REQ) OTL(Robot.CMD) ,[XIC(Robot.CMD) XIC(RobotInputs.ib_Running) ,XIO(RobotInputs.ib_Running) EQ(RobotInputs.iW_PositionEcho,AOI_RobotPos.Barcode) ] ADD(OP220_Seq.CurrentStep,10,OP220_Seq.NextStep) OTU(Robot.CMD) ];
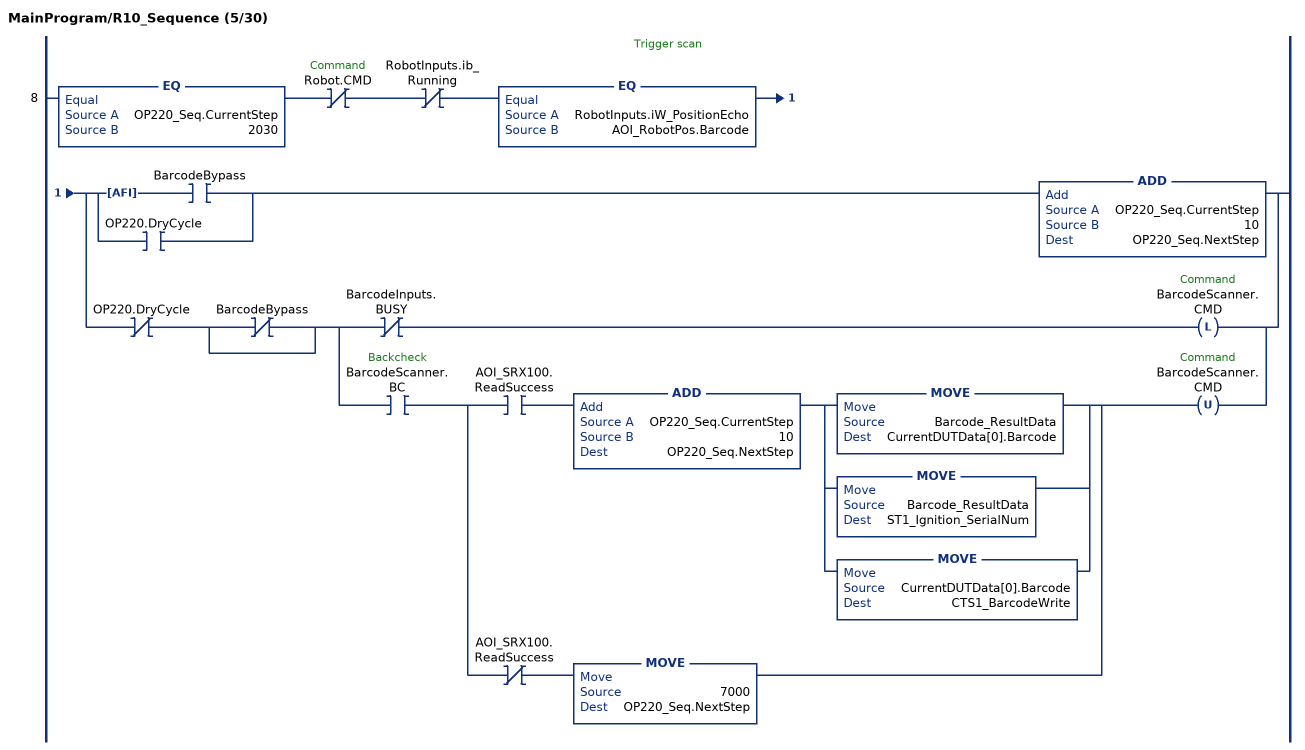
   // Trigger scan
   8: EQ(OP220_Seq.CurrentStep,2030)XIO(Robot.CMD)XIO(RobotInputs.ib_Running)EQ(RobotInputs.iW_PositionEcho,AOI_RobotPos.Barcode)[[AFI() XIC(BarcodeBypass) ,XIC(OP220.DryCycle) ] ADD(OP220_Seq.CurrentStep,10,OP220_Seq.NextStep) ,XIO(OP220.DryCycle) [XIO(BarcodeBypass) ,] [XIO(BarcodeInputs.BUSY) OTL(BarcodeScanner.CMD) ,XIC(BarcodeScanner.BC) [XIC(AOI_SRX100.ReadSuccess) ADD(OP220_Seq.CurrentStep,10,OP220_Seq.NextStep) [MOVE(Barcode_ResultData,CurrentDUTData[0].Barcode) ,[MOVE(Barcode_ResultData,ST1_Ignition_SerialNum) ,MOVE(CurrentDUTData[0].Barcode,CTS1_BarcodeWrite) ] ] ,XIO(AOI_SRX100.ReadSuccess) MOVE(7000,OP220_Seq.NextStep) ] OTU(BarcodeScanner.CMD) ] ];
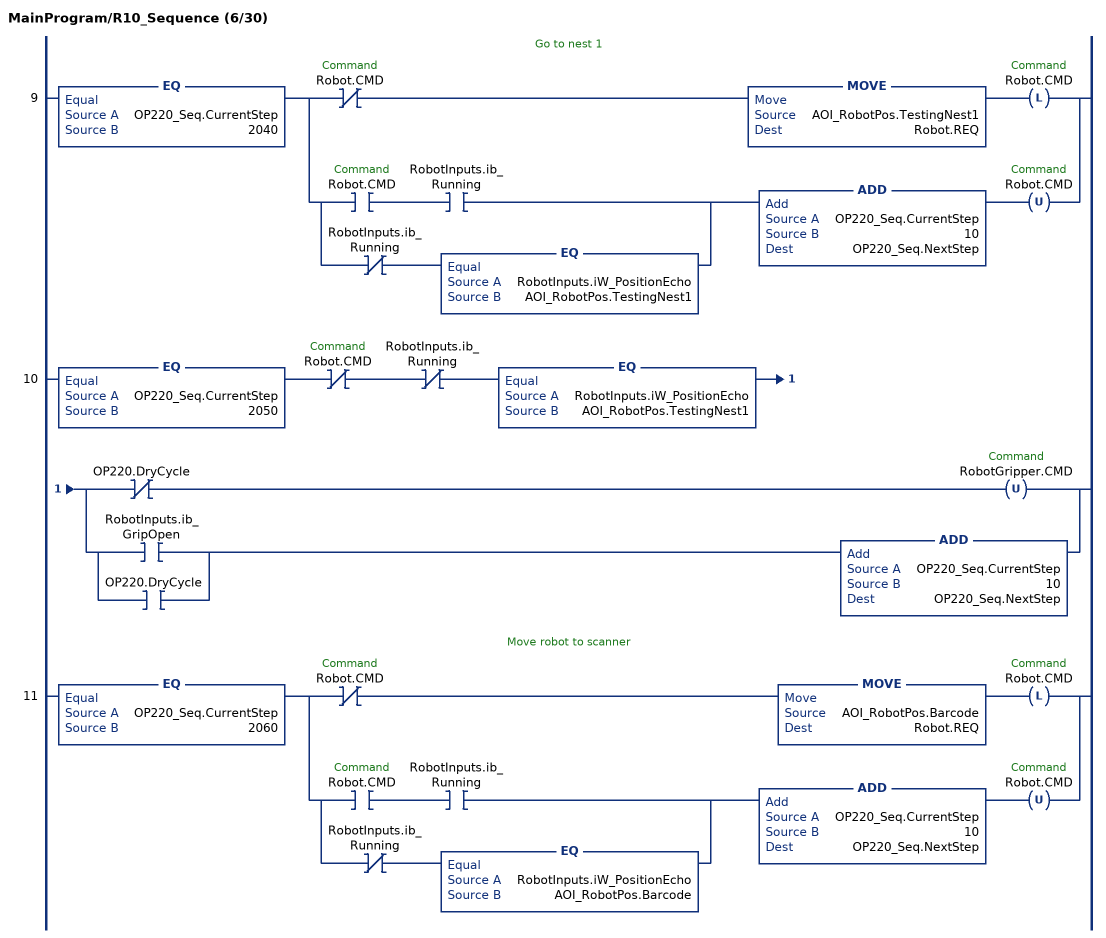
   // Go to nest 1
   9: EQ(OP220_Seq.CurrentStep,2040)[XIO(Robot.CMD) MOVE(AOI_RobotPos.TestingNest1,Robot.REQ) OTL(Robot.CMD) ,[XIC(Robot.CMD) XIC(RobotInputs.ib_Running) ,XIO(RobotInputs.ib_Running) EQ(RobotInputs.iW_PositionEcho,AOI_RobotPos.TestingNest1) ] ADD(OP220_Seq.CurrentStep,10,OP220_Seq.NextStep) OTU(Robot.CMD) ];
   10: EQ(OP220_Seq.CurrentStep,2050)XIO(Robot.CMD)XIO(RobotInputs.ib_Running)EQ(RobotInputs.iW_PositionEcho,AOI_RobotPos.TestingNest1)[XIO(OP220.DryCycle) OTU(RobotGripper.CMD) ,[XIC(RobotInputs.ib_GripOpen) ,XIC(OP220.DryCycle) ] ADD(OP220_Seq.CurrentStep,10,OP220_Seq.NextStep) ];
   // Move robot to scanner
   11: EQ(OP220_Seq.CurrentStep,2060)[XIO(Robot.CMD) MOVE(AOI_RobotPos.Barcode,Robot.REQ) OTL(Robot.CMD) ,[XIC(Robot.CMD) XIC(RobotInputs.ib_Running) ,XIO(RobotInputs.ib_Running) EQ(RobotInputs.iW_PositionEcho,AOI_RobotPos.Barcode) ] ADD(OP220_Seq.CurrentStep,10,OP220_Seq.NextStep) OTU(Robot.CMD) ];
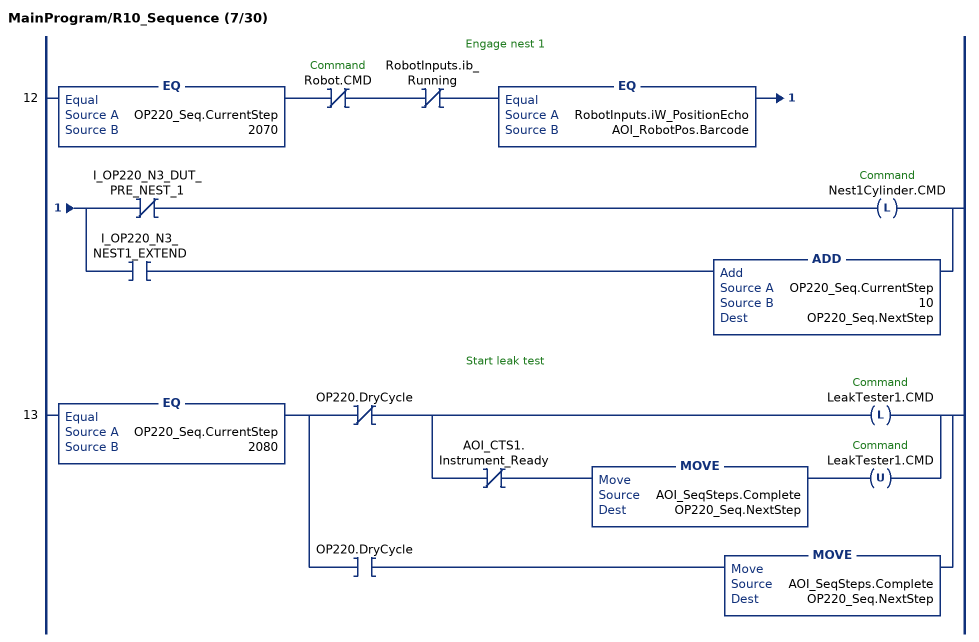
   // Engage nest 1
   12: EQ(OP220_Seq.CurrentStep,2070)XIO(Robot.CMD)XIO(RobotInputs.ib_Running)EQ(RobotInputs.iW_PositionEcho,AOI_RobotPos.Barcode)[XIO(I_OP220_N3_DUT_PRE_NEST_1) OTL(Nest1Cylinder.CMD) ,XIC(I_OP220_N3_NEST1_EXTEND) ADD(OP220_Seq.CurrentStep,10,OP220_Seq.NextStep) ];
   // Start leak test
   13: EQ(OP220_Seq.CurrentStep,2080)[XIO(OP220.DryCycle) [OTL(LeakTester1.CMD) ,XIO(AOI_CTS1.Instrument_Ready) MOVE(AOI_SeqSteps.Complete,OP220_Seq.NextStep) OTU(LeakTester1.CMD) ] ,XIC(OP220.DryCycle) MOVE(AOI_SeqSteps.Complete,OP220_Seq.NextStep) ];
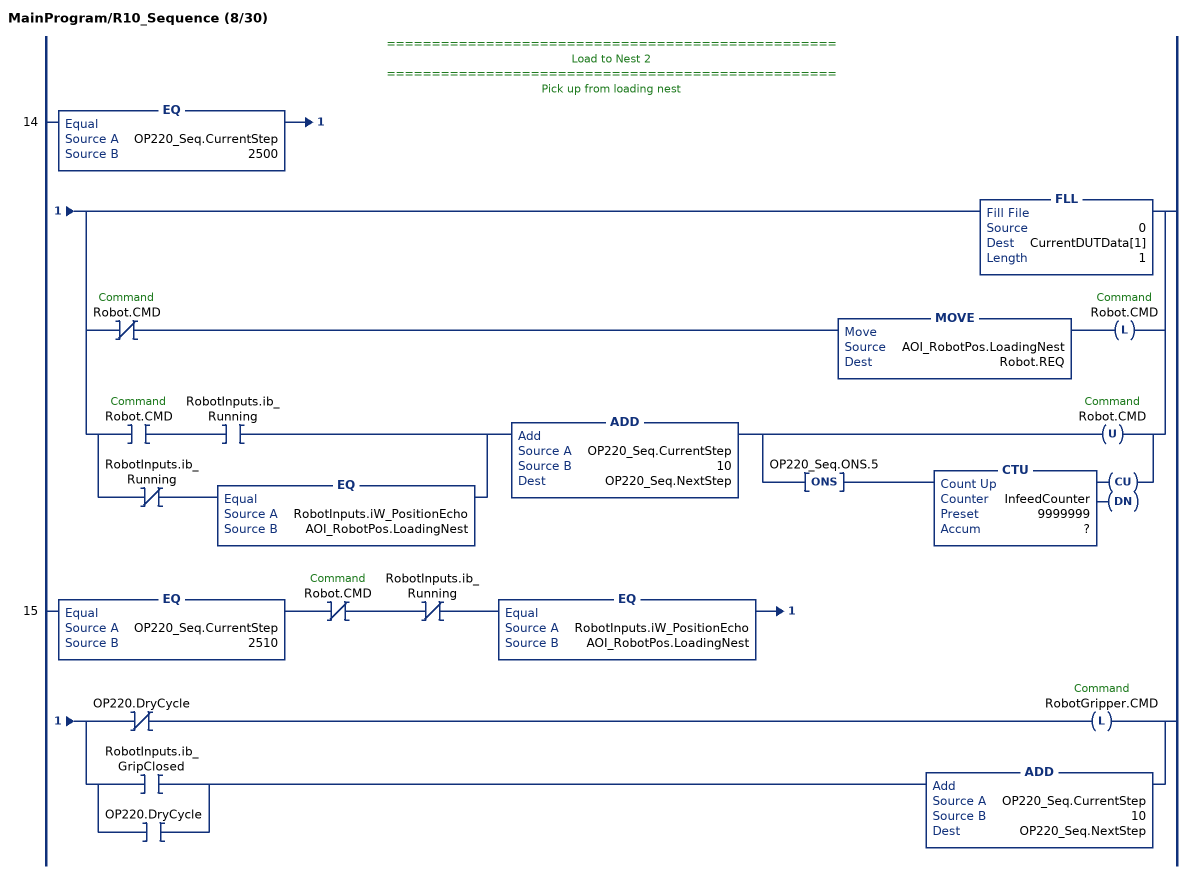
   // ==================================================
   // Load to Nest 2
   // ==================================================
   // Pick up from loading nest
   14: EQ(OP220_Seq.CurrentStep,2500)[FLL(0,CurrentDUTData[1],1) ,XIO(Robot.CMD) MOVE(AOI_RobotPos.LoadingNest,Robot.REQ) OTL(Robot.CMD) ,[XIC(Robot.CMD) XIC(RobotInputs.ib_Running) ,XIO(RobotInputs.ib_Running) EQ(RobotInputs.iW_PositionEcho,AOI_RobotPos.LoadingNest) ] ADD(OP220_Seq.CurrentStep,10,OP220_Seq.NextStep) [OTU(Robot.CMD) ,ONS(OP220_Seq.ONS.5) CTU(InfeedCounter,?,?) ] ];
   15: EQ(OP220_Seq.CurrentStep,2510)XIO(Robot.CMD)XIO(RobotInputs.ib_Running)EQ(RobotInputs.iW_PositionEcho,AOI_RobotPos.LoadingNest)[XIO(OP220.DryCycle) OTL(RobotGripper.CMD) ,[XIC(RobotInputs.ib_GripClosed) ,XIC(OP220.DryCycle) ] ADD(OP220_Seq.CurrentStep,10,OP220_Seq.NextStep) ];
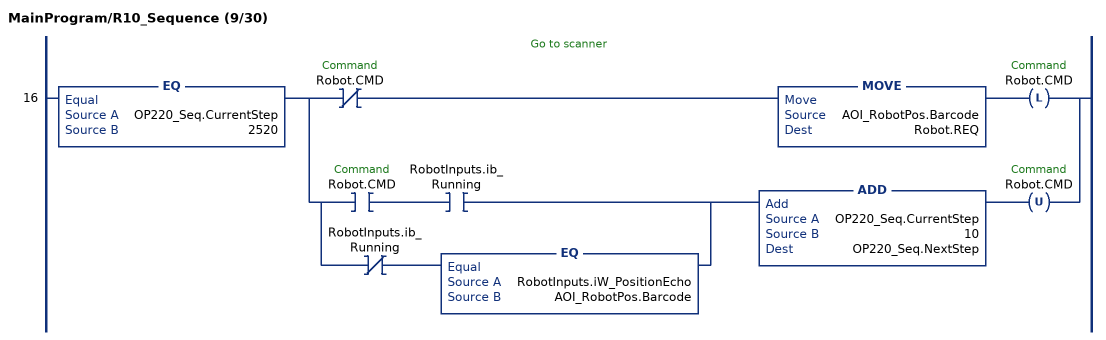
   // Go to scanner
   16: EQ(OP220_Seq.CurrentStep,2520)[XIO(Robot.CMD) MOVE(AOI_RobotPos.Barcode,Robot.REQ) OTL(Robot.CMD) ,[XIC(Robot.CMD) XIC(RobotInputs.ib_Running) ,XIO(RobotInputs.ib_Running) EQ(RobotInputs.iW_PositionEcho,AOI_RobotPos.Barcode) ] ADD(OP220_Seq.CurrentStep,10,OP220_Seq.NextStep) OTU(Robot.CMD) ];
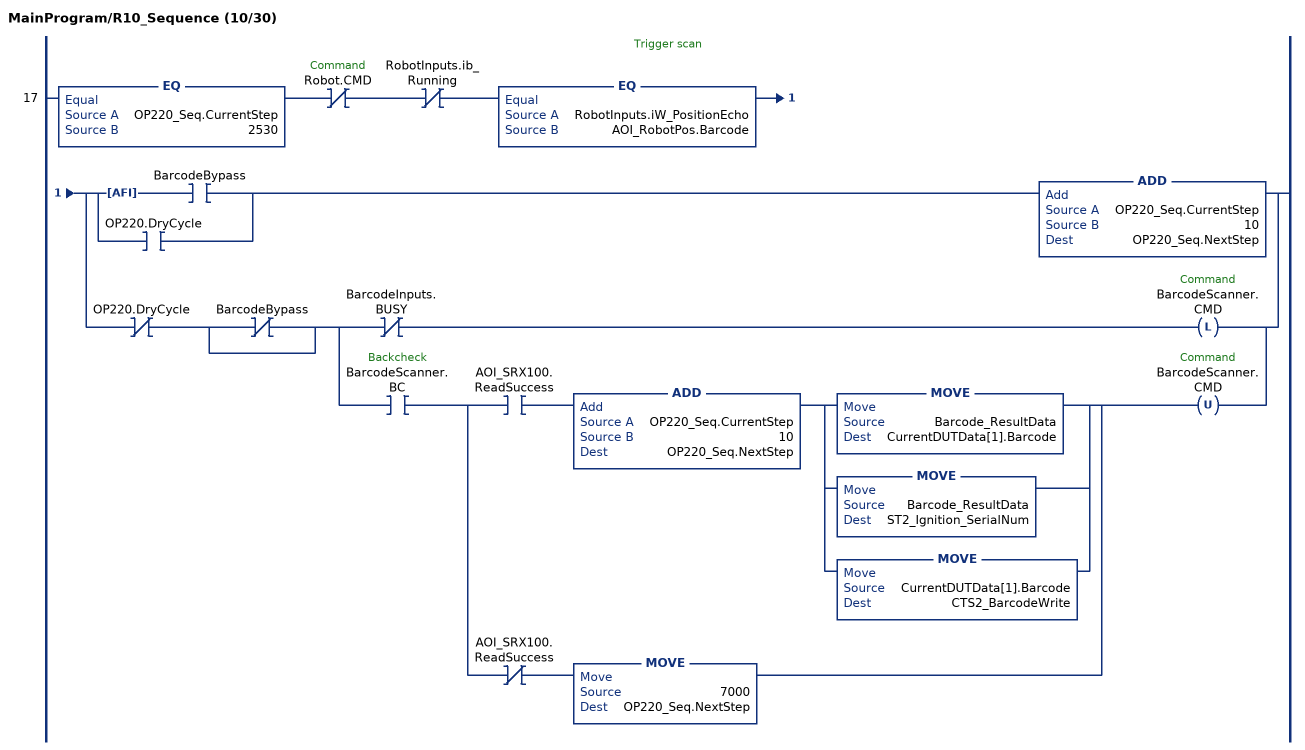
   // Trigger scan
   17: EQ(OP220_Seq.CurrentStep,2530)XIO(Robot.CMD)XIO(RobotInputs.ib_Running)EQ(RobotInputs.iW_PositionEcho,AOI_RobotPos.Barcode)[[AFI() XIC(BarcodeBypass) ,XIC(OP220.DryCycle) ] ADD(OP220_Seq.CurrentStep,10,OP220_Seq.NextStep) ,XIO(OP220.DryCycle) [XIO(BarcodeBypass) ,] [XIO(BarcodeInputs.BUSY) OTL(BarcodeScanner.CMD) ,XIC(BarcodeScanner.BC) [XIC(AOI_SRX100.ReadSuccess) ADD(OP220_Seq.CurrentStep,10,OP220_Seq.NextStep) [MOVE(Barcode_ResultData,CurrentDUTData[1].Barcode) ,[MOVE(Barcode_ResultData,ST2_Ignition_SerialNum) ,MOVE(CurrentDUTData[1].Barcode,CTS2_BarcodeWrite) ] ] ,XIO(AOI_SRX100.ReadSuccess) MOVE(7000,OP220_Seq.NextStep) ] OTU(BarcodeScanner.CMD) ] ];
